# EPICS autosave request: iocBoot/ioc14ida/auto_settings.req
14IDA:DAC1_4.VAL
# 14IDA:DAC1_1.VAL
14IDA:DAC1_2.VAL
14IDA:DAC1_3.VAL

#file "mono_pid_control_settings.req",   P=14IDA:, PID=mono_pid1
#file "saveData_settings.req",          P=14IDA:
file "CARS_16_motor_settings.req",      P=14IDA:
file "HeatLoadShutter.req",             P=14IDA:,Q=HLS
file "UndPos.req",                      P=14IDA:,Q=Und
###############
#file "DAC_AMVE-9210_settings.req "      P=14IDA:,DAC=DAC1
#file "VME_DAC_settings.req",             P=14IDA:,DAC=DAC1
#14IDA:DAC1_4.VAL
